Staubli VAL3: libload.pgx

program libload(string s_Item (dimensions=1))
begin
  pub:libLoad(s_Item)
  call pub:main()
end
